% RSLogix 500 project HOURMETER.RSS, saved by version 8.30.00.16 %
PROJECT "UNTITLED"    % processor: Bul.1763 MicroLogix 1100 Series B %

PROGRAM FILES
  LAD 2   8 rungs

DATA FILES
  O0 OUTPUT  4 elements
  I1 INPUT  6 elements
  S2 STATUS  66 elements
  B3 BINARY  1 elements
  T4 TIMER  2 elements
  C5 COUNTER  1 elements
  R6 CONTROL  1 elements
  N7 INTEGER  4 elements
  F8 FLOAT  1 elements

LADDER 2
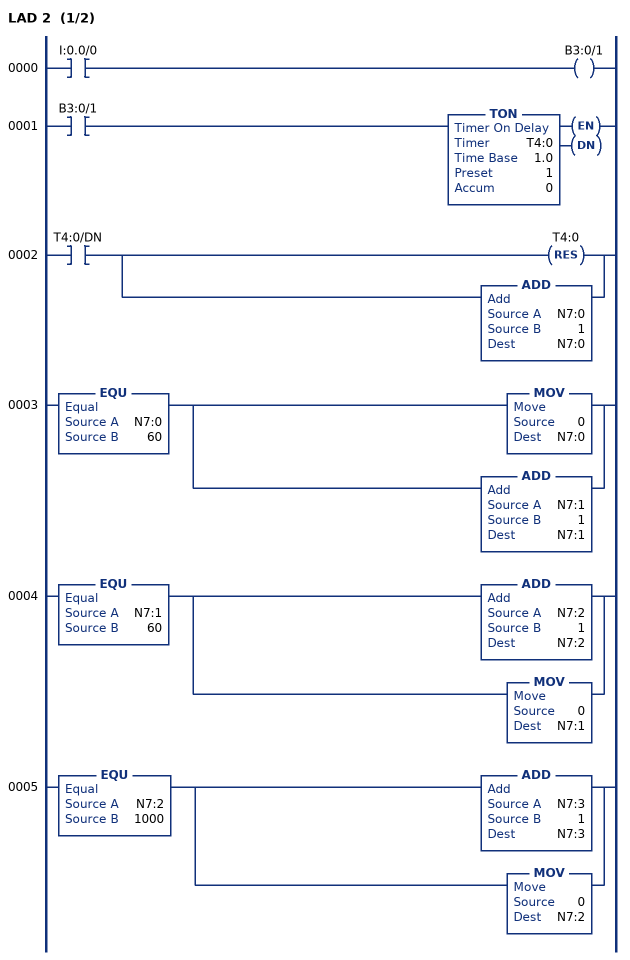
% Rung: 0 %
SOR XIC I:0.0/0 OTE B3:0/1 EOR
% Rung: 1 %
SOR XIC B3:0/1 TON T4:0 1.0 1 0 EOR
% Rung: 2 %
SOR XIC T4:0/DN BST RES T4:0 NXB ADD N7:0 1 N7:0 BND EOR
% Rung: 3 %
SOR EQU N7:0 60 BST MOV 0 N7:0 NXB ADD N7:1 1 N7:1 BND EOR
% Rung: 4 %
SOR EQU N7:1 60 BST ADD N7:2 1 N7:2 NXB MOV 0 N7:1 BND EOR
% Rung: 5 %
SOR EQU N7:2 1000 BST ADD N7:3 1 N7:3 NXB MOV 0 N7:2 BND EOR

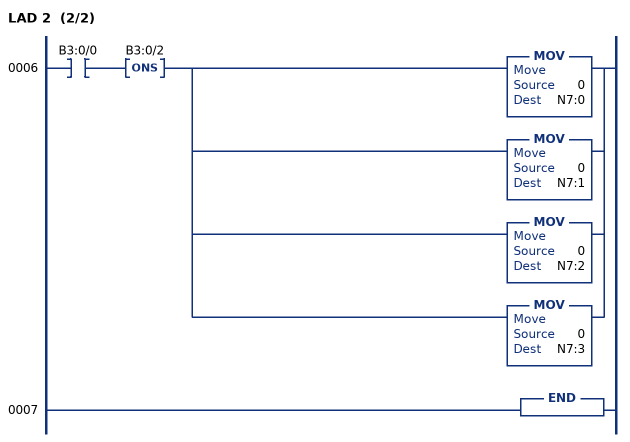
% Rung: 6 %
SOR XIC B3:0/0 ONS B3:0/2 BST MOV 0 N7:0 NXB MOV 0 N7:1 NXB MOV 0 N7:2 NXB MOV 0 N7:3 BND EOR
% Rung: 7 %
SOR END EOR

DATA TABLE (non-zero values as saved)
DATA B3
% B3:0 % 0X0007
DATA T4
% .PRE .ACC %
% T4:0 % 1 0
% T4:1 % 60 0
DATA N7
% N7:0 % 16 0 0 0
